TYPE hmiAlarms_TypeStruct :
STRUCT

	slitter : hmiAlarmsSlitter_TypeStruct;
	rotaryKnife : hmiAlarmsRotaryKnife_TypeStruct;
	lowerStacker	: hmiAlarmsSimpleStacker_TypeStruct;
	upperStacker	: hmiAlarmsComplexStacker_TypeStruct;

END_STRUCT
END_TYPE

(* stored: Version 1.1.0.1
   DUT hmiAlarms_TypeStruct: Id {155311ad-f558-4c7f-afed-ad26b5e924a8} *)
